// TIA Portal V16 export
// export: Created 2021-09-08T12:46:12.1803129Z, ExportSetting WithDefaults, DisplayName Totally Integrated Automation Portal, DisplayVersion V16 Update 3, DisplayName TIA Portal Version Control Interface, DisplayVersion V16 Update 2, DisplayName TIA Portal Openness, DisplayVersion V16 Update 3, DisplayName TIA Portal Teamcenter Gateway, DisplayVersion V16, DisplayName STEP 7 Professional, DisplayVersion V16 Update 3, DisplayName STEP 7 Safety, DisplayVersion V16, DisplayName WinCC Advanced, DisplayVersion V16 Update 3
DATA_BLOCK "AllPump_DB"   // DB9
VERSION : 0.1
// stored: AutoNumber true, DBAccessibleFromOPCUA true, InstanceOfName AllPump, InstanceOfType FB
"AllPump"
   // VAR
   //    PU30x { S7_SetPoint := 'True'} : "PumpCntrl2Pu1Fc";
   //    cmUZ_P30x { S7_SetPoint := 'True'} : Bool;
   //    cmUZ_P120x : Bool;
   //    cmUZ_P150x : Bool;
   //    tmrLowPresP30x { S7_SetPoint := 'True'} : TON_TIME;
   //    tmrLowFreqP30x { S7_SetPoint := 'True'} : TON_TIME;
   //    tLowPresP30x { S7_SetPoint := 'True'} : Time;
   //    tLowFreqP30x : Time;
   //    PU120x { S7_SetPoint := 'True'} : "PumpCntrl2Pu1Fc";
   //    tmrLowPresP120x { S7_SetPoint := 'True'} : TON_TIME;
   //    tLowPresP120x { S7_SetPoint := 'True'} : Time;
   //    tNoPulseP120x : Time;
   //    PU150x { S7_SetPoint := 'True'} : "PumpCntrl2Pu1Fc";
   //    tmrLowPresP150x { S7_SetPoint := 'True'} : TON_TIME;
   //    tLowPresP150x { S7_SetPoint := 'True'} : Time;
   //    tNoPulseP150x : Time;
   //    noPulseTOF_P120x { S7_SetPoint := 'True'} : "noPulseTOF";
   //    noPulseTOF_P150x { S7_SetPoint := 'True'} : "noPulseTOF";
   //    P701 { S7_SetPoint := 'True'} : "PumpCntr";
   //    P702 { S7_SetPoint := 'True'} : "PumpCntr";
   //    P901 { S7_SetPoint := 'True'} : "PumpCntr";
   //    P1301 { S7_SetPoint := 'True'} : "PumpCntr";
   //    P2001 { S7_SetPoint := 'True'} : "PumpCntr";
   //    C501 { S7_SetPoint := 'True'} : "PumpCntr";
   //    sel2pu_P70x { S7_SetPoint := 'True'} : "sel2pu";
   // END_VAR
BEGIN
END_DATA_BLOCK
